// TIA Portal project "testeControleNivel" (V16)
// teste stl para exemplo de controle de nivel de tanque

(* hardware
DEVICE "S7-1200 station_1"  S7-1200 Station
   slot 0: "Rack_0"  S7-1200 Rack  Rack  V1.0
   slot 1: "PLC_1"  CPU 1215C DC/DC/DC  6ES7 215-1AG40-0XB0  V4.4
*)

// ===== PLC "PLC_1"  CPU 1215C DC/DC/DC =====

VAR_GLOBAL   // PLC tag table "Default tag table"
   "pb1" AT %I0.0 : Bool;
   "pb2" AT %I0.1 : Bool;
   "high" AT %I0.2 : Bool;
   "low" AT %I0.3 : Bool;
   "stop" AT %I0.4 : Bool;
   "fill" AT %Q0.0 : Bool;
   "drain" AT %Q0.1 : Bool;
END_VAR

FUNCTION "Block_1" : Void   // FC1, SCL
{ S7_Optimized_Access := 'TRUE' }
VERSION : 0.1
   VAR_INPUT
      PB1 : Bool;   // push botton Fill
      PB2 : Bool;   // push botton Drain
      HIGH : Bool;   // sensor de nivel alto
      LOW : Bool;   // sensor de nivel baixo
      STOP : Bool;   // emergencia
   END_VAR
   VAR_OUTPUT
      FILL : Bool;   // Encher
      DRAIN : Bool;   // Esvaziar
   END_VAR
BEGIN
   (*IF (#PB1 OR #FILL AND #STOP) AND NOT #HIGH THEN
       #FILL := TRUE;
   ELSE
       #FILL := FALSE;

   END_IF;

   IF (#PB2 OR #DRAIN AND #STOP AND #LOW) THEN
       #DRAIN:=TRUE;
   ELSE
       #DRAIN := FALSE;

   END_IF; *)

   //forma resumida
   //#FILL := (#PB1 OR #FILL) AND NOT #STOP AND NOT #HIGH;
   //#DRAIN := (#PB2 OR #DRAIN) AND NOT #STOP AND NOT #LOW;
   //
   (* =========================
      CONTROLE DE ENCHIMENTO
      ========================= *)

   IF (#PB1 OR #FILL) AND NOT #STOP AND NOT #HIGH THEN
       #FILL := TRUE;
   ELSE
       #FILL := FALSE;
   END_IF;


   (* =========================
      CONTROLE DE DRENAGEM
      ========================= *)

   IF (#PB2 OR #DRAIN) AND NOT #STOP AND #LOW THEN
       #DRAIN := TRUE;
   ELSE
       #DRAIN := FALSE;
   END_IF;
END_FUNCTION

ORGANIZATION_BLOCK "Main"   // OB1, LAD, ProgramCycle
TITLE = "Main Program Sweep (Cycle)"
{ S7_Optimized_Access := 'TRUE' }
VERSION : 0.1
   VAR_INPUT
      Initial_Call : Bool;   // Initial call of this OB
      Remanence : Bool;   // =True, if remanent data are available
   END_VAR
BEGIN

REGION Network 1: FC1 Controle de nivel
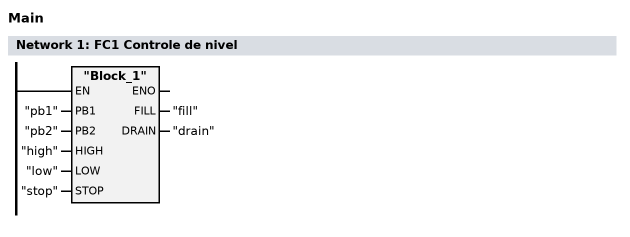
   RUNG wire#powerrail
      "Block_1"(PB1 := "pb1", PB2 := "pb2", HIGH := "high", LOW := "low", STOP := "stop", FILL => "fill", DRAIN => "drain")
   END_RUNG
   // the same network as SCL:
   "Block_1"(PB1 := "pb1",
             PB2 := "pb2",
             HIGH := "high",
             LOW := "low",
             STOP := "stop",
             FILL => "fill",
             DRAIN => "drain");
END_REGION
END_ORGANIZATION_BLOCK